(* CoDeSys 2.3.9.28 project: aula16.pro *)
(* Libraries: Standard.lib 27.1.09 11:27:38, Util.lib 27.1.09 11:27:38, IecSfc.lib 24.11.08 08:07:15, SysLibTime.lib 27.1.09 11:27:38, SysTaskInfo.lib 24.11.08 08:07:15, SYSLIBCALLBACK.LIB 27.1.09 11:27:38 *)

(* PLC configuration (modules and I/O channels)
CPX-CEC [Root] node -1, in %IB0 out %QB0 {StringParam = 2773,0,0,0,0; ByteParam = 0; ByteParam = 31; ByteParam = 0; ByteParam = 0; ByteParam = 0; ByteParam = 0; ByteParam = 0; ByteParam = 0; ByteParam = 2; ByteParam = 0; ByteParam = 0; ByteParam = 0; ByteParam = 32; ByteParam = 0; ByteParam = 0; ByteParam = 5; ByteParam = 0; ByteParam = 0; ByteParam = 0; ByteParam = 0; ByteParam = 0; ByteParam = 0; ByteParam = 0; ByteParam = 0; ByteParam = 14; ByteParam = 240; ByteParam = 192; ByteParam = 168; ByteParam = 2; ByteParam = 10; ByteParam = 255; ByteParam = 255; ByteParam = 0; ByteParam = 0; ByteParam = 192; ByteParam = 168; ByteParam = 1; ByteParam = 1; ByteParam = 192; ByteParam = 168; ByteParam = 2; ByteParam = 10; ByteParam = 255; ByteParam = 255; ByteParam = 0; ByteParam = 0; ByteParam = 192; ByteParam = 168; ByteParam = 1; ByteParam = 1}
  Hexswitch AT %IB0 [HexSwitch] rotary switch 0 = STOP, 1-15 = RUN
  IOModules [CPX_MASTER] node 0, in %IB4 out %QB0
*)

(* Global variable list: Global_Variables *)
VAR_GLOBAL

	START: BOOL;
	STOP: BOOL;

	LP: BOOL;
	SP: BOOL;

	A: BOOL;
	B: BOOL;

	C1: BOOL;
	C2: BOOL;
	C3: BOOL;

	T1 : TON;
	T2 : TON;
	T3 : TON;
	T4 : TON;

	ROBO : ROBO;
	CONT1 : CTU;

	ME: BOOL;
	MD: BOOL;
	MS: BOOL;
	MDE: BOOL;

	AROB:BOOL;
	RROB:BOOL;

	MEM1: BOOL;
	MEM2: BOOL;
	MEM3: BOOL;
	MEM4: BOOL;

	MEMSTART:BOOL;
	MEMSTOP: BOOL;

	MEM_INI: BOOL;
	MEMC1: BOOL;
	MEMC3: BOOL;

END_VAR

(* POU PLC_PRG, ST *)
PROGRAM PLC_PRG
VAR

END_VAR
T1(IN:=NOT T2.Q,PT:=T#1S);
T2(IN:=T1.Q AND CONT1.Q ,PT:=T#1S);
T3(IN:=B, PT:=T#5S);
T4(IN:=CONT1.Q, PT:=T#10S);

ROBO(ENTRADA:= AROB);
CONT1(CU:= ME AND C1 AND MEM_INI, RESET:= STOP OR T4.Q, PV:= 3);



IF NOT MEM_INI AND START THEN
	MEMSTART:=TRUE;
END_IF


IF NOT MEM_INI AND MEMSTART THEN
	ME:=TRUE;

	IF C1 THEN
		ME:=FALSE;
		MEM_INI:=TRUE;
		MEMSTART:=FALSE;
	END_IF

END_IF


IF MEM_INI THEN

	IF NOT MEMSTOP THEN

		IF START OR MEM4 THEN
			MEM1:=TRUE;
			MEM4:=FALSE;

			MEMSTART:=TRUE;
		END_IF


		IF C1 AND MEM1 AND NOT RROB THEN
			MEM1:=FALSE;

			AROB:=TRUE;
			MEMC1:=TRUE;
		END_IF


		IF ROBO.SAIDA THEN
			AROB:=FALSE;
			RROB:=TRUE;
		END_IF


		IF RROB AND MEMC1 THEN
			MEM2:=TRUE;

			MEMC1:=FALSE;
			MD:=TRUE;
			RROB:=FALSE;
		END_IF


		IF C2 AND MEM2 THEN
			MEM2:=FALSE;

			MD:=FALSE;
			MDE:=TRUE;
		END_IF


		IF B THEN
			MDE:=FALSE;
		END_IF


		IF T3.Q THEN
			MS:=TRUE;
		END_IF


		IF A AND MS THEN
			MEM3:=TRUE;

			MS:=FALSE;
			MD:=TRUE;
		END_IF


		IF C3 AND MEM3 THEN
			MEM3:=FALSE;

			MD:=FALSE;
			AROB:=TRUE;
			MEMC3:=TRUE;
		END_IF


		IF RROB AND MEMC3 THEN
			ME:=TRUE;
			RROB:=FALSE;
			MEMC3:=FALSE;
		END_IF


		IF C1 AND ME THEN
			ME:=FALSE;
			IF MEMSTART AND NOT MEMSTOP THEN
				MEM4:=TRUE;
			END_IF
		END_IF


		IF CONT1.Q AND NOT T4.Q THEN
			LP := T1.Q;
			MEM4:=FALSE;
		END_IF


		IF T4.Q THEN
			LP:=FALSE;
		END_IF


	ELSE
		IF C1 AND A THEN
			MEMSTOP:=FALSE;
		END_IF


		IF C1 THEN
			ME:=FALSE;
		END_IF


		IF A THEN
			MS:=FALSE;
		END_IF

	END_IF
END_IF


IF STOP THEN

	MEMSTOP:=TRUE;

	ME:=TRUE;
	MD:=FALSE;
	MS:=TRUE;
	MDE:=FALSE;

	MEM4:=FALSE;
	LP:=FALSE;

END_IF
END_PROGRAM

(* POU ROBO, ST *)
FUNCTION_BLOCK ROBO
VAR_INPUT
	ENTRADA:BOOL;
END_VAR
VAR_OUTPUT
	SAIDA:BOOL;
END_VAR
VAR
	T1_ROBO : TON;
END_VAR
T1_ROBO(IN:= ENTRADA, PT:=T#2S);

IF T1_ROBO.Q THEN
	SAIDA := TRUE;
ELSE
	SAIDA := FALSE;
END_IF
END_FUNCTION_BLOCK

(* POU PISCA_LED, ST *)
FUNCTION_BLOCK PISCA_LED
VAR_INPUT
	LIGA : BOOL;
	DESLIGA : BOOL;
END_VAR
VAR_OUTPUT
	SAIDA : BOOL;
END_VAR
VAR
	T1 : TON;
	T2 : TON;
	MEM : BOOL;
END_VAR
T1(IN:=LP, PT:=T#1S);
T2(IN:= NOT LP, PT:=T#1S);

IF LIGA AND T1.Q AND NOT MEM THEN
	LP := FALSE;
END_IF


IF NOT LIGA AND  T2.Q AND NOT MEM THEN
	LP := TRUE;
END_IF


IF DESLIGA THEN
	MEM := TRUE;
END_IF

IF LIGA THEN
	MEM := FALSE;
END_IF
END_FUNCTION_BLOCK

(* Visualisation screen
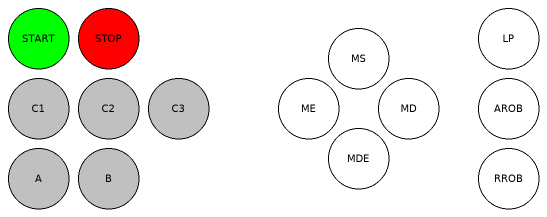
ellipse at (50,120)-(111,181): text "C1"; alarm colour if C1; toggles C1
ellipse at (120,120)-(181,181): text "C2"; alarm colour if C2; toggles C2
ellipse at (190,120)-(251,181): text "C3"; alarm colour if C3; toggles C3
ellipse at (50,50)-(111,111): text "START"; alarm colour if START; taps START
ellipse at (120,50)-(181,111): text "STOP"; alarm colour if STOP; taps STOP
ellipse at (320,120)-(381,181): text "ME"; alarm colour if ME
ellipse at (370,70)-(431,131): text "MS"; alarm colour if MS
ellipse at (370,170)-(431,231): text "MDE"; alarm colour if MDE
ellipse at (420,120)-(481,181): text "MD"; alarm colour if MD
ellipse at (520,50)-(581,111): text "LP"; alarm colour if LP
ellipse at (50,190)-(111,251): text "A"; alarm colour if A; toggles A
ellipse at (120,190)-(181,251): text "B"; alarm colour if B; toggles B
ellipse at (520,120)-(581,181): text "AROB"; alarm colour if AROB
ellipse at (520,190)-(581,251): text "RROB"; alarm colour if RROB
*)
